FUNCTION_BLOCK _LWORD_TestSuite EXTENDS TcUnit.FB_TestSuite
VAR
END_VAR

TestAddress();
TestClearReference();
TestClone();
TestTypeNameReturnsExpected();
TestIsFloat();
TestIsSigned();
TestMakeReferenceToFollowsReference();
TestMakeReferenceToUpdatesReference();
TestSize();
TestValueReturnsExpectedAfterInit();
TestValueReturnsExpectedAfterChange();
TestSerializeTypeWith();
TestSerializeWith();
TestTryDeserializeFrom();
TestTryMakeReferenceToFollowsReference();
TestTryMakeReferenceToUpdatesReference();

METHOD PUBLIC TestAddress
VAR
    _type : _LWORD(0);
    notExpected : PVOID := 0;
    actual : PVOID;
END_VAR
TEST('TestAddress');

actual := _type.Address;

AssertFalse(
    Condition := (notExpected = actual),
    Message := 'Type did not return a valid address.'
);

TEST_FINISHED();
END_METHOD

METHOD PUBLIC TestClearReference
VAR
    _type : _LWORD(0);
	target : LWORD := 0;
    expected : LWORD := 0;
    actual : LWORD;
END_VAR
TEST('TestClearReference');

_type.MakeReferenceTo(target);
_type.ClearReference();
target := 123;

actual := _type.Value;

AssertEquals(
    Expected := expected,
    Actual := actual,
    Message := 'Value incorrectly followed target change'
);

TEST_FINISHED();
END_METHOD

METHOD PUBLIC TestClone
VAR
    _type : _LWORD(123);
	clone : I_Datatype;
	isValidClone : BOOL;
	compareResult : DINT;
END_VAR
TEST('TestClone');

clone := _type.Clone();

isValidClone := clone <> 0;

IF isValidClone THEN
	compareResult := memcmp(_type.Address, clone.Address, clone.Size);
END_IF

AssertTrue(
	Condition := isValidClone,
	Message := 'Clone did not produce a clone'
);

AssertEquals_DINT(
	Expected := 0,
    Actual := compareResult,
    Message := 'Clone did not return a valid clone.'
);

clone.Dispose();

TEST_FINISHED();
END_METHOD

METHOD PUBLIC TestIsFloat
VAR
    _type : _LWORD(0);
END_VAR
TEST('TestIsFloat');

AssertFalse(
	Condition := _type.IsFloat,
    Message := 'Type did not correctly identify itself as being unsigned'
);

TEST_FINISHED();
END_METHOD

METHOD PUBLIC TestIsSigned
VAR
    _type : _LWORD(0);
END_VAR
TEST('TestIsSigned');

AssertFalse(
	Condition := _type.IsSigned,
    Message := 'Type did not correctly identify itself as being unsigned'
);

TEST_FINISHED();
END_METHOD

METHOD PUBLIC TestMakeReferenceToFollowsReference
VAR
    _type : _LWORD(0);
	target : LWORD := 0;
    expected : LWORD := 123;
    actual : LWORD;
END_VAR
TEST('TestMakeReferenceToFollowsReference');

_type.MakeReferenceTo(target);
target := 123;

actual := _type.Value;

AssertEquals(
    Expected := expected,
    Actual := actual,
    Message := 'Value did not follow target change'
);

TEST_FINISHED();
END_METHOD

METHOD PUBLIC TestMakeReferenceToUpdatesReference
VAR
    _type : _LWORD(0);
	target : LWORD := 0;
    expected : LWORD := 123;
    actual : LWORD;
END_VAR
TEST('TestMakeReferenceToUpdatesReference');

_type.MakeReferenceTo(target);
_type.Value := 123;

actual := target;

AssertEquals(
    Expected := expected,
    Actual := actual,
    Message := 'Value did not update target'
);

TEST_FINISHED();
END_METHOD

METHOD PUBLIC TestSerializeTypeWith
VAR
    _type : _LWORD(0);
    serializer : JsonSerializer;
    expected : STRING(500) := '{"typeName":"LWORD","minValue":0,"maxValue":18446744073709551615,"isSigned":false,"isFloat":false}';
    actual : STRING(500);
END_VAR
TEST('TestSerializeTypeWith');

serializer.Reset();
_type.SerializeTypeWith(serializer);
serializer.TryGetSerializedData(ADR(actual), SIZEOF(actual));

AssertEquals_STRING(
    Expected := expected,
    Actual := actual,
    Message := 'Serialization of type did not return correct string.'
);

TEST_FINISHED();
END_METHOD

METHOD PUBLIC TestSerializeWith
VAR
    _type : _LWORD(65535);
    serializer : JsonSerializer;
    expected : STRING := '65535';
    actual : STRING(500);
END_VAR
TEST('TestSerializeWith');

serializer.Reset();
_type.SerializeWith(serializer);
serializer.TryGetSerializedData(ADR(actual), SIZEOF(actual));

AssertEquals_STRING(
    Expected := expected,
    Actual := actual,
    Message := 'Serialization of type data did not return correct string.'
);

TEST_FINISHED();
END_METHOD

METHOD PUBLIC TestSize
VAR
    _type : _LWORD(0);
    expected : UDINT := SIZEOF(LWORD);
    actual : UDINT;
END_VAR
TEST('TestSize');

actual := _type.Size;

AssertEquals_UDINT(
    Expected := Expected,
    Actual := actual,
    Message := 'Type did not return the correct size.'
);

TEST_FINISHED();
END_METHOD

METHOD PUBLIC TestTryDeserializeFrom
VAR
    deserializer : JsonDeserializer;
    feedback : DeserializerFeedback;
    json : STRING := '65535';
    _type : _LWORD(0);
    expected : LWORD := 65535;
    actual : LWORD;
 END_VAR
TEST('TestTryDeserializeFrom');

deserializer.Reset();
deserializer.TryLoad(json);
_type.TryDeserializeFrom(Deserializer, Feedback);

actual := _type.Value;

AssertEquals(
    Expected := expected,
    Actual := actual,
    Message := 'Type did not deserialize correctly.'
);

TEST_FINISHED();
END_METHOD

METHOD PUBLIC TestTryMakeReferenceToFollowsReference
VAR
    _type : _LWORD(0);
	target : _LWORD(0);
    expected : LWORD := 123;
    actual : LWORD;
END_VAR
TEST('TestTryMakeReferenceToFollowsReference');

_type.TryMakeReferenceTo(target);
target.Value := 123;

actual := _type.Value;

AssertEquals(
    Expected := expected,
    Actual := actual,
    Message := 'Value did not follow target change'
);

TEST_FINISHED();
END_METHOD

METHOD PUBLIC TestTryMakeReferenceToUpdatesReference
VAR
    _type : _LWORD(0);
	target : _LWORD(0);
    expected : LWORD := 123;
    actual : LWORD;
END_VAR
TEST('TestTryMakeReferenceToUpdatesReference');

_type.TryMakeReferenceTo(target);
_type.Value := 123;

actual := target.Value;

AssertEquals(
    Expected := expected,
    Actual := actual,
    Message := 'Value did not update target'
);

TEST_FINISHED();
END_METHOD

METHOD PUBLIC TestTypeNameReturnsExpected
VAR
    _type : _LWORD(0);
    expected : STRING := 'LWORD';
    actual : STRING;
END_VAR
TEST('TestTypeNameReturnsExpected');

actual := _type.TypeName;

AssertEquals_STRING(
    Expected := expected,
    Actual := actual,
    Message := 'Type did not return correct iec type.'
);

TEST_FINISHED();
END_METHOD

METHOD PUBLIC TestValueReturnsExpectedAfterChange
VAR
    _type : _LWORD(0);
    expected : LWORD := 65535;
    actual : LWORD;
END_VAR
TEST('TestValueReturnsExpectedAfterChange');

_type.Value := 65535;

actual := _type.Value;

AssertEquals(
    Expected := expected,
    Actual := actual,
    Message := 'Expected value not returned after change.'
);

TEST_FINISHED();
END_METHOD

METHOD PUBLIC TestValueReturnsExpectedAfterInit
VAR
    _type : _LWORD(65535);
    expected : LWORD := 65535;
    actual : LWORD;
END_VAR
TEST('TestValueReturnsExpectedAfterInit');

actual := _type.Value;

AssertEquals(
    Expected := expected,
    Actual := actual,
    Message := 'Expected value not returned after Init.'
);

TEST_FINISHED();
END_METHOD

END_FUNCTION_BLOCK

(* stored: Version 1.1.0.1, ProductVersion 3.1.4024.12
   POU _LWORD_TestSuite: Id {8bee7435-0cc3-01ef-36d2-2fa7a4bcaa7d}, SpecialFunc None
   Method TestAddress: Id {20513951-c889-0e41-3d88-d1d5e2a53596}
   Method TestClearReference: Id {a6202762-e3b8-032a-1af5-063da5587975}
   Method TestClone: Id {52f6cfa7-a44c-02e6-3775-d8fab9fbac81}
   Method TestIsFloat: Id {c95934c0-f79f-41f8-9b63-d1898f37634b}
   Method TestIsSigned: Id {700c4700-0114-0281-0609-85500d620172}
   Method TestMakeReferenceToFollowsReference: Id {ddcc3124-ac3e-024b-2c96-44248b17bbfa}
   Method TestMakeReferenceToUpdatesReference: Id {3cbd1f6c-f58c-0dc4-3265-6e3b4cf475c5}
   Method TestSerializeTypeWith: Id {293bf8b1-6ef8-03dc-3e92-c79c34e5a1a3}
   Method TestSerializeWith: Id {c3ba1401-90c5-06cd-345d-c2dfa00f6264}
   Method TestSize: Id {ead8a0d7-cc35-01b0-03bc-a1e73e9402e9}
   Method TestTryDeserializeFrom: Id {4df9ae53-4f19-0d2e-2f2a-ce375a5e4685}
   Method TestTryMakeReferenceToFollowsReference: Id {1b80c11f-944b-0f1c-2dbc-b6f182df91e6}
   Method TestTryMakeReferenceToUpdatesReference: Id {694b42df-7a35-0a01-28dc-4bbc2378508a}
   Method TestTypeNameReturnsExpected: Id {f06b4d20-5bd6-01db-0b60-ae5f39583122}
   Method TestValueReturnsExpectedAfterChange: Id {514a7432-0fa7-0181-1cae-46014dcfcdc0}
   Method TestValueReturnsExpectedAfterInit: Id {f2f69751-0b49-0b3f-0744-d4522472d532} *)
